FUNCTION_BLOCK Drive2 EXTENDS DriveBase
VAR_INPUT
END_VAR
VAR_OUTPUT
END_VAR
VAR
END_VAR

{error 'Add method implementation or delete method to use base implementation'}
METHOD Disable : BOOL
END_METHOD

{error 'Add method implementation or delete method to use base implementation'}
METHOD Enable : BOOL
END_METHOD

END_FUNCTION_BLOCK

(* stored: Version 1.1.0.1
   POU Drive2: Id {90361d04-0b47-48c1-82d5-1e635a3bf13e}, SpecialFunc None
   Method Disable: Id {0cd07071-3cf6-4d23-8a8b-4df48e1911fd}
   Method Enable: Id {d20e2793-f759-4988-9dba-d99d6c67cf04} *)
